FUNCTION_BLOCK AE_AX_SERVER_0_CLIENT_1_0 (* Receive a remote OPC-UA method call via SERVER_0 and write the resulting state back via CLIENT_1_0, driven by an AE_AX bidirectional adapter Plug (1 Event forward, state back) *)
  (* Standard: 61499-2; Description: Copyright (c) 2026 HR Agrartechnik GmbH This program and the accompanying materials are made available under the terms of the Eclipse Public License 2.0 which is available at https://www.eclipse.org/legal/epl-2.0/ SPDX-License-Identifier: EPL-2.0 *)
  (* Version 1.0, 2026-09-03, Franz Höpfinger, HR Agrartechnik GmbH, initial API and implementation and/or initial documentation *)
  PACKAGE adapter::net;
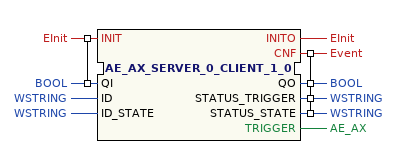
  EVENT_INPUT
    INIT : EInit WITH QI; (* Initialization *)
  END_EVENT
  EVENT_OUTPUT
    INITO : EInit; (* Initialization Confirm *)
    CNF WITH QO, STATUS_TRIGGER, STATUS_STATE; (* QO/STATUS updated *)
  END_EVENT
  VAR_INPUT
    QI : BOOL;
    ID : WSTRING; (* Lokale Methodenadresse (ACTION=CREATE_METHOD) fuer den Trigger-Methodenaufruf *)
    ID_STATE : WSTRING; (* Remote-Ziel-Adresse (ACTION=WRITE) fuer den Zustand *)
  END_VAR
  VAR_OUTPUT
    QO : BOOL; (* TRUE nur wenn SERVER_0_1 und STATE_CLIENT aktuell beide QO=TRUE melden *)
    STATUS_TRIGGER : WSTRING; (* STATUS von SERVER_0_1 *)
    STATUS_STATE : WSTRING; (* STATUS von STATE_CLIENT *)
  END_VAR
  PLUGS
    TRIGGER : adapter::types::bidirectional::AE_AX; (* Trigger (in), Zustand (out) *)
  END_PLUGS
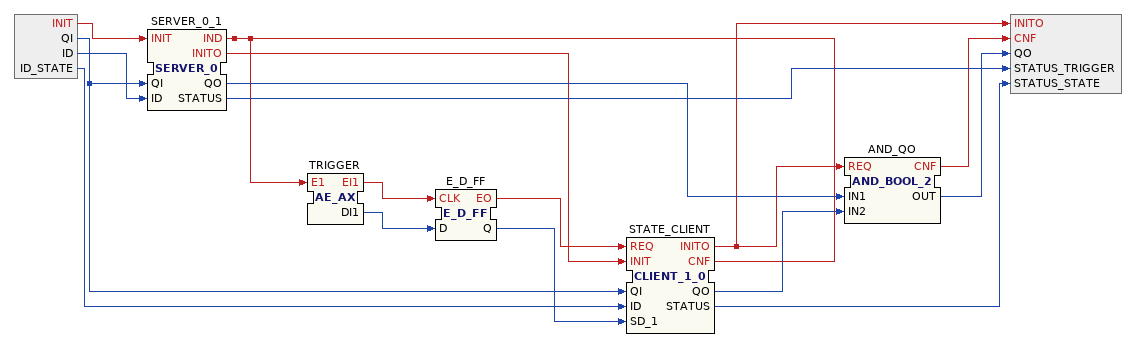
  FBS
    SERVER_0_1 : iec61499::net::SERVER_0;
    E_D_FF : iec61499::events::E_D_FF;
    STATE_CLIENT : iec61499::net::CLIENT_1_0;
    AND_QO : iec61131::booleanOperators::AND_BOOL_2;
  END_FBS
  EVENT_CONNECTIONS
    INIT TO SERVER_0_1.INIT;
    STATE_CLIENT.INITO TO INITO;
    STATE_CLIENT.INITO TO AND_QO.REQ;
    SERVER_0_1.IND TO TRIGGER.E1;
    TRIGGER.EI1 TO E_D_FF.CLK;
    E_D_FF.EO TO STATE_CLIENT.REQ;
    SERVER_0_1.INITO TO STATE_CLIENT.INIT;
    SERVER_0_1.IND TO AND_QO.REQ;
    STATE_CLIENT.CNF TO AND_QO.REQ;
    AND_QO.CNF TO CNF;
  END_CONNECTIONS
  DATA_CONNECTIONS
    QI TO SERVER_0_1.QI;
    QI TO STATE_CLIENT.QI;
    ID TO SERVER_0_1.ID;
    ID_STATE TO STATE_CLIENT.ID;
    TRIGGER.DI1 TO E_D_FF.D;
    E_D_FF.Q TO STATE_CLIENT.SD_1;
    SERVER_0_1.QO TO AND_QO.IN1;
    STATE_CLIENT.QO TO AND_QO.IN2;
    AND_QO.OUT TO QO;
    SERVER_0_1.STATUS TO STATUS_TRIGGER;
    STATE_CLIENT.STATUS TO STATUS_STATE;
  END_CONNECTIONS
END_FUNCTION_BLOCK
